TYPE "ValveMachine_Config"
VERSION : 0.1
// Block: ValveMachine_Config
   STRUCT
      DelayPressureRunningTimeout : Time;
      DelayMissingCondition : Time;
      Rest_LsQty : Int;
      Work_LsQty : Int;
      Rest_RetainAut : Bool;
      Work_RetainAut : Bool;
      V : ValveConfig;
   END_STRUCT;

END_TYPE
